TYPE ST_CoolingSystemGet :
STRUCT
	CoolingSystemMode		:	eConditioningStates;
	HeatPumpStatus			: 	eHeatPumpState;
	CoolantTemperature		:	REAL;
	CoolantPressure			:	REAL;
	EnclosureDewpoint		:	REAL;
		
	
	HeatPumpSystemGet 		: REFERENCE TO ST_HeatpumpSystemGet;	
	Events					: ST_CoolingSystemEvents;
END_STRUCT
END_TYPE

(* stored: Version 1.1.0.1, ProductVersion 3.1.4024.12
   DUT ST_CoolingSystemGet: Id {c5f9e8e4-f620-4cbc-bb65-ad5a08f7db42} *)
